// TIA Portal project "TrapanoFB" (V16)

(* hardware
DEVICE "S7-1200 station_1"  S7-1200 Station
   slot 0: "Telaio di montaggio_0"  S7-1200 Rack  Rack  V1.0
   slot 1: "PLC_1"  CPU 1214C DC/DC/DC  6ES7 214-1AG40-0XB0  V4.1
*)

// ===== PLC "PLC_1"  CPU 1214C DC/DC/DC =====

VAR_GLOBAL   // PLC tag table "Tabella delle variabili standard"
   "START" AT %I0.0 : Bool;
   "A" AT %I0.1 : Bool;
   "B" AT %I0.2 : Bool;
   "M" AT %I0.3 : Bool;
   "X" AT %I0.4 : Bool;
   "Y" AT %I0.5 : Bool;
   "DOWN" AT %Q0.0 : Bool;
   "UP" AT %Q0.1 : Bool;
   "ROTATE" AT %Q0.2 : Bool;
   "OIL" AT %Q0.3 : Bool;
END_VAR

VAR_GLOBAL CONSTANT   // PLC tag table "Tabella delle variabili standard"
   "TEMPO_TRASCORSO" : Time := T#5s;
END_VAR

DATA_BLOCK "Trapano_DB"   // DB1
{ S7_Optimized_Access := 'TRUE' }
VERSION : 0.1
// stored: InstanceOfName Trapano
"Trapano"
BEGIN
END_DATA_BLOCK

FUNCTION_BLOCK "Trapano"   // FB1, LAD
{ S7_Optimized_Access := 'TRUE' }
VERSION : 0.1
   VAR_INPUT
      START : Bool;
      "A" : Bool;
      "B" : Bool;
      "M" : Bool;
      X : Bool;
      Y : Bool;
      TEMPO_TRASCORSO : Time := T#5s;
   END_VAR
   VAR_OUTPUT
      Down : Bool;
      Up : Bool;
      Rotate : Bool;
      Oil : Bool;
   END_VAR
   VAR RETAIN
      Home : Bool := true;
      Scendi : Bool;
      Pezzo_Alto : Bool;
      Pezzo_Alto_Risalita : Bool;
      Lubrifica : Bool;
      Foro : Bool;
      Sali : Bool;
      Wait : Bool;
   END_VAR
   VAR
      IEC_Timer_0_Instance : TON_TIME;
   END_VAR
   VAR_TEMP   // added for the SCL form of the ladder/FBD networks
      _w1 : Bool;
   END_VAR
BEGIN

REGION Network 1
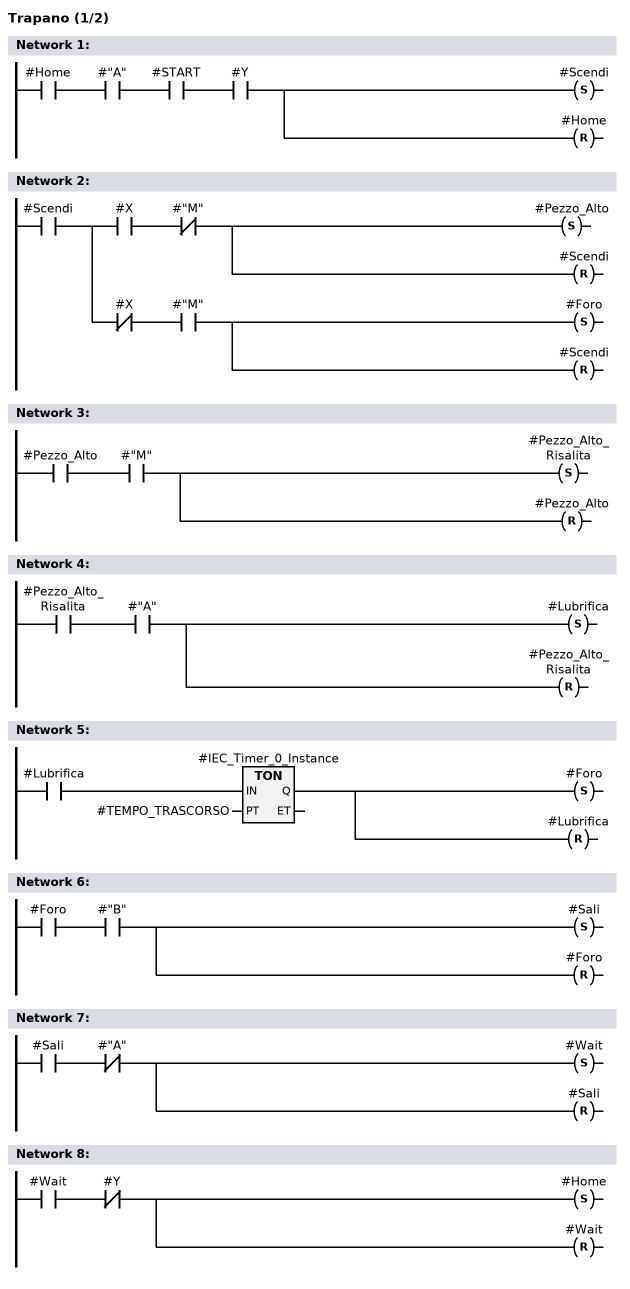
   RUNG wire#powerrail
      Contact( #Home )
      Contact( #"A" )
      Contact( #START )
      Contact( #Y )
      wire#w1
      S_Coil( #Scendi )
   END_RUNG
   RUNG wire#w1
      R_Coil( #Home )
   END_RUNG
   // the same network as SCL:
   IF #Home AND #"A" AND #START AND #Y THEN
       #Scendi := TRUE;
       #Home := FALSE;
   END_IF;
END_REGION

REGION Network 2
   RUNG wire#powerrail
      Contact( #Scendi )
      wire#w1
      Contact( #X )
      I_Contact( #"M" )
      wire#w2
      S_Coil( #Pezzo_Alto )
   END_RUNG
   RUNG wire#w2
      R_Coil( #Scendi )
   END_RUNG
   RUNG wire#w1
      I_Contact( #X )
      Contact( #"M" )
      wire#w3
      S_Coil( #Foro )
   END_RUNG
   RUNG wire#w3
      R_Coil( #Scendi )
   END_RUNG
   // the same network as SCL:
   IF #Scendi AND #X AND NOT #"M" THEN #Pezzo_Alto := TRUE; END_IF;
   #_w1 := #Scendi;
   IF #Scendi AND #X AND NOT #"M" THEN #Scendi := FALSE; END_IF;
   IF #_w1 AND NOT #X AND #"M" THEN
       #Foro := TRUE;
       #Scendi := FALSE;
   END_IF;
END_REGION

REGION Network 3
   RUNG wire#powerrail
      Contact( #Pezzo_Alto )
      Contact( #"M" )
      wire#w1
      S_Coil( #Pezzo_Alto_Risalita )
   END_RUNG
   RUNG wire#w1
      R_Coil( #Pezzo_Alto )
   END_RUNG
   // the same network as SCL:
   IF #Pezzo_Alto AND #"M" THEN
       #Pezzo_Alto_Risalita := TRUE;
       #Pezzo_Alto := FALSE;
   END_IF;
END_REGION

REGION Network 4
   RUNG wire#powerrail
      Contact( #Pezzo_Alto_Risalita )
      Contact( #"A" )
      wire#w1
      S_Coil( #Lubrifica )
   END_RUNG
   RUNG wire#w1
      R_Coil( #Pezzo_Alto_Risalita )
   END_RUNG
   // the same network as SCL:
   IF #Pezzo_Alto_Risalita AND #"A" THEN
       #Lubrifica := TRUE;
       #Pezzo_Alto_Risalita := FALSE;
   END_IF;
END_REGION

REGION Network 5
   #IEC_Timer_0_Instance(IN := #Lubrifica, PT := #TEMPO_TRASCORSO);   // TON
   IF #IEC_Timer_0_Instance.Q THEN
       #Foro := TRUE;
       #Lubrifica := FALSE;
   END_IF;
END_REGION

REGION Network 6
   RUNG wire#powerrail
      Contact( #Foro )
      Contact( #"B" )
      wire#w1
      S_Coil( #Sali )
   END_RUNG
   RUNG wire#w1
      R_Coil( #Foro )
   END_RUNG
   // the same network as SCL:
   IF #Foro AND #"B" THEN
       #Sali := TRUE;
       #Foro := FALSE;
   END_IF;
END_REGION

REGION Network 7
   RUNG wire#powerrail
      Contact( #Sali )
      I_Contact( #"A" )
      wire#w1
      S_Coil( #Wait )
   END_RUNG
   RUNG wire#w1
      R_Coil( #Sali )
   END_RUNG
   // the same network as SCL:
   IF #Sali AND NOT #"A" THEN
       #Wait := TRUE;
       #Sali := FALSE;
   END_IF;
END_REGION

REGION Network 8
   RUNG wire#powerrail
      Contact( #Wait )
      I_Contact( #Y )
      wire#w1
      S_Coil( #Home )
   END_RUNG
   RUNG wire#w1
      R_Coil( #Wait )
   END_RUNG
   // the same network as SCL:
   IF #Wait AND NOT #Y THEN
       #Home := TRUE;
       #Wait := FALSE;
   END_IF;
END_REGION

REGION Network 9
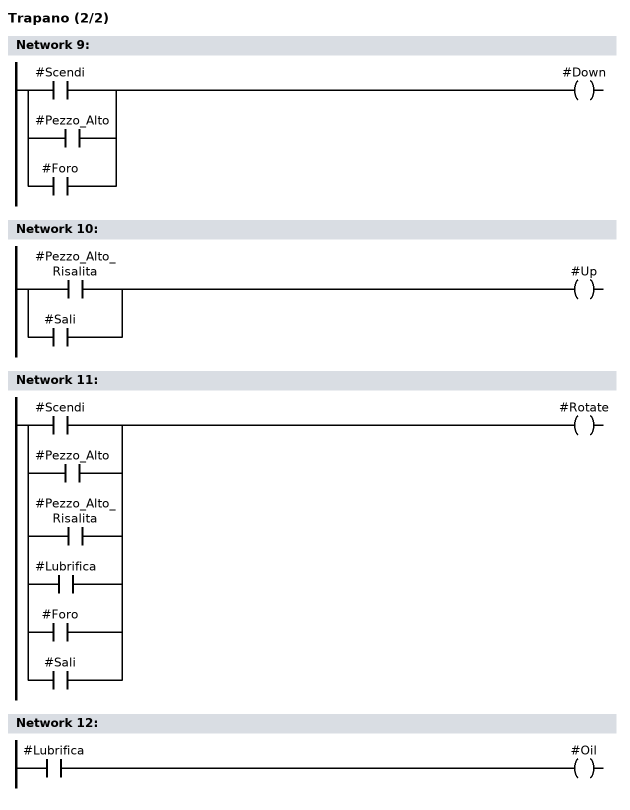
   RUNG wire#powerrail
      Contact( #Scendi )
      wire#w1
      Coil( #Down )
   END_RUNG
   RUNG wire#powerrail
      Contact( #Pezzo_Alto )
   END_RUNG wire#w1
   RUNG wire#powerrail
      Contact( #Foro )
   END_RUNG wire#w1
   // the same network as SCL:
   #Down := #Scendi OR #Pezzo_Alto OR #Foro;
END_REGION

REGION Network 10
   RUNG wire#powerrail
      Contact( #Pezzo_Alto_Risalita )
      wire#w1
      Coil( #Up )
   END_RUNG
   RUNG wire#powerrail
      Contact( #Sali )
   END_RUNG wire#w1
   // the same network as SCL:
   #Up := #Pezzo_Alto_Risalita OR #Sali;
END_REGION

REGION Network 11
   RUNG wire#powerrail
      Contact( #Scendi )
      wire#w1
      Coil( #Rotate )
   END_RUNG
   RUNG wire#powerrail
      Contact( #Pezzo_Alto )
   END_RUNG wire#w1
   RUNG wire#powerrail
      Contact( #Pezzo_Alto_Risalita )
   END_RUNG wire#w1
   RUNG wire#powerrail
      Contact( #Lubrifica )
   END_RUNG wire#w1
   RUNG wire#powerrail
      Contact( #Foro )
   END_RUNG wire#w1
   RUNG wire#powerrail
      Contact( #Sali )
   END_RUNG wire#w1
   // the same network as SCL:
   #Rotate := #Scendi OR #Pezzo_Alto OR #Pezzo_Alto_Risalita OR #Lubrifica OR #Foro OR #Sali;
END_REGION

REGION Network 12
   RUNG wire#powerrail
      Contact( #Lubrifica )
      Coil( #Oil )
   END_RUNG
   // the same network as SCL:
   #Oil := #Lubrifica;
END_REGION
END_FUNCTION_BLOCK

ORGANIZATION_BLOCK "Main"   // OB1, LAD, ProgramCycle
TITLE = "Main Program Sweep (Cycle)"
{ S7_Optimized_Access := 'TRUE' }
VERSION : 0.1
   VAR_INPUT
      Initial_Call : Bool;   // Initial call of this OB
      Remanence : Bool;   // =True, if remanent data are available
   END_VAR
BEGIN

REGION Network 1
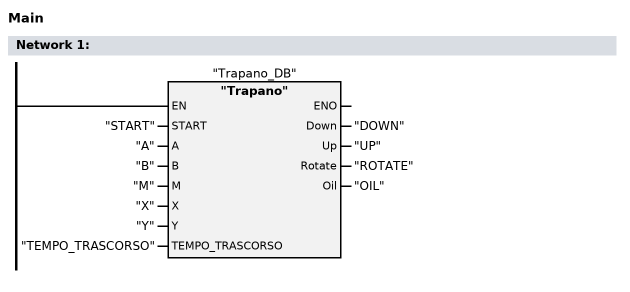
   RUNG wire#powerrail
      "Trapano_DB"(START := "START", "A" := "A", "B" := "B", "M" := "M", X := "X", Y := "Y", TEMPO_TRASCORSO := "TEMPO_TRASCORSO", Down => "DOWN", Up => "UP", Rotate => "ROTATE", Oil => "OIL")
   END_RUNG
   // the same network as SCL:
   "Trapano_DB"(START := "START",   // "Trapano"
                "A" := "A",
                "B" := "B",
                "M" := "M",
                X := "X",
                Y := "Y",
                TEMPO_TRASCORSO := "TEMPO_TRASCORSO",
                Down => "DOWN",
                Up => "UP",
                Rotate => "ROTATE",
                Oil => "OIL");
END_REGION
END_ORGANIZATION_BLOCK